FUNCTION_BLOCK StandardSection
  (* Standard: 61499-2 *)
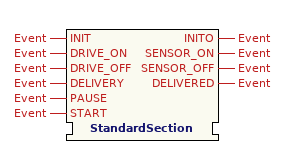
  EVENT_INPUT
    INIT;
    DRIVE_ON;
    DRIVE_OFF;
    DELIVERY;
    PAUSE;
    START;
  END_EVENT
  EVENT_OUTPUT
    INITO;
    SENSOR_ON;
    SENSOR_OFF;
    DELIVERED;
  END_EVENT
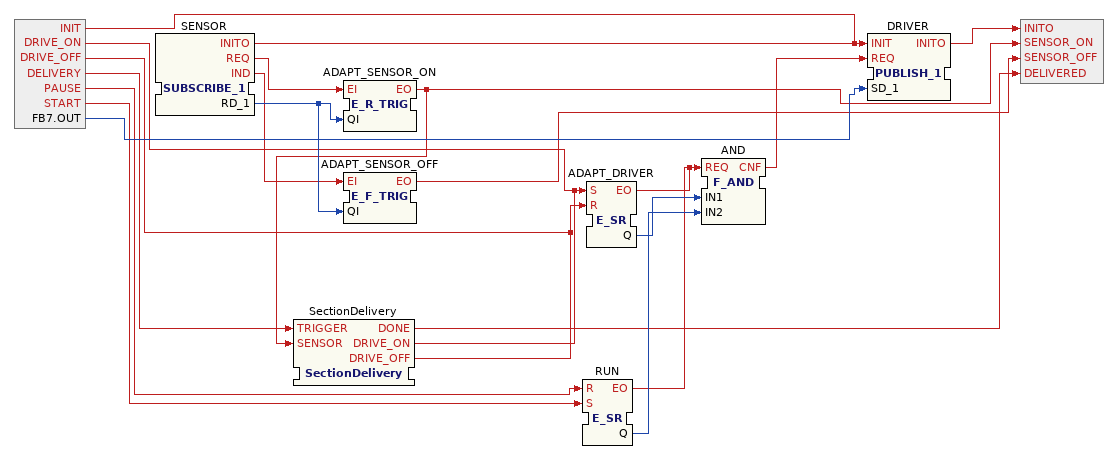
  FBS
    DRIVER : PUBLISH_1;
    SENSOR : SUBSCRIBE_1;
    ADAPT_DRIVER : E_SR;
    ADAPT_SENSOR_ON : E_R_TRIG;
    ADAPT_SENSOR_OFF : E_F_TRIG;
    SectionDelivery : SectionDelivery;
    AND : F_AND;
    RUN : E_SR;
  END_FBS
  EVENT_CONNECTIONS
    INIT TO DRIVER.INIT;
    DRIVER.INITO TO INITO;
    SENSOR.INITO TO DRIVER.INIT;
    ADAPT_DRIVER.EO TO AND.REQ;
    DRIVE_ON TO ADAPT_DRIVER.S;
    DRIVE_OFF TO ADAPT_DRIVER.R;
    SENSOR.REQ TO ADAPT_SENSOR_ON.EI;
    ADAPT_SENSOR_ON.EO TO SENSOR_ON;
    ADAPT_SENSOR_OFF.EO TO SENSOR_OFF;
    SENSOR.IND TO ADAPT_SENSOR_OFF.EI;
    DELIVERY TO SectionDelivery.TRIGGER;
    SectionDelivery.DRIVE_ON TO ADAPT_DRIVER.S;
    SectionDelivery.DRIVE_OFF TO ADAPT_DRIVER.R;
    ADAPT_SENSOR_ON.EO TO SectionDelivery.SENSOR;
    SectionDelivery.DONE TO DELIVERED;
    PAUSE TO RUN.R;
    START TO RUN.S;
    RUN.EO TO AND.REQ;
    AND.CNF TO DRIVER.REQ;
  END_CONNECTIONS
  DATA_CONNECTIONS
    ADAPT_DRIVER.Q TO AND.IN1;
    SENSOR.RD_1 TO ADAPT_SENSOR_ON.QI;
    SENSOR.RD_1 TO ADAPT_SENSOR_OFF.QI;
    RUN.Q TO AND.IN2;
    FB7.OUT TO DRIVER.SD_1;
  END_CONNECTIONS
END_FUNCTION_BLOCK
